RoboDK station: inspeccion2.rdk

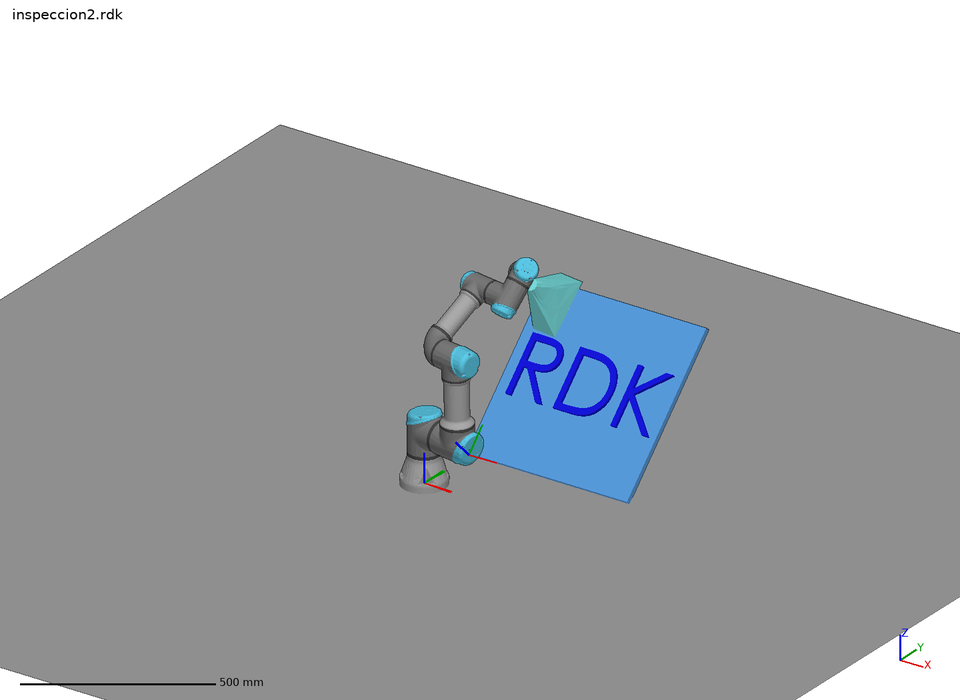
[picture v0: the station drawn from its stored meshes, robots at their saved joint values, targets as dots, program paths as lines]
Station inspeccion2 (saved by RoboDK 5.7.3). Poses are relative to the parent item; angles as X-Y-Z fixed-axis rotations.
  - frame UR3e Base at (0, 0, 0) mm, rotated rx 0 ry 0 rz -3.41 deg
    - robot UR3e: 6 axes, payload 3 kg, reach 500 mm, repeatability 0.03 mm, weight 11 kg
        modified DH rows (alpha deg, a mm, theta deg, d mm): 0, 0, 0, 151.9; 90, 0, 180, 0; 0, 243.55, 0, 0; 0, 213.2, 0, 131.05; -90, 0, 0, 85.35; 90, 0, 180, 92.1
        joint limits [-360, -360, -360, -360, -360, -360] to [360, 360, 360, 360, 360, 360]; home [0, -90, -90, 0, 90, 0]; saved at [83.892, -88.327, -60.278, -74.725, 133.683, -2.499]
      - tool Camera 2, TCP at (0, 0, 0) mm, size 104.4 x 65.1 x 142.2 mm
      - tool Camera view, TCP at (0, 0, 0) mm, size 136.1 x 159.8 x 161.7 mm
  - frame Suelo at (0, 0, 0) mm
    - object Floor at (0, 0, 0) mm, size 3000 x 3000 x 0 mm, geometry from Floor.sld
  - frame Frame 3 at (0, 200, 0) mm, rotated rx 45 ry 0 rz 0 deg
    - object RoboDK RDK Plate 100x100mm at (0, 0, 0) mm, size 500 x 500 x 25 mm, geometry from RoboDK-RDK-Plate-100x100mm.sld
